{attribute addProperty BoxType "EL2258-0000-0016"}
{attribute addProperty Id "MTO_Inputs_ChannelAT %I*ARRAY[0..7] OF MTO_Inputs_Channel_5AD475AF8721090MTO_Outputs_10x_ChannelAT %Q*ARRAY[0..7] OF MTO_Outputs_10x_Channel_4C67AB5F45845730WcStateAT %I*WcState_F855686C1620InfoDataAT %I*InfoData_0BDED7BF144180"}
{attribute addProperty CRC "3021902586"}
{attribute addProperty SizeInBites "5616"}
{attribute addProperty SizeInBytes "702"}
TYPE EL2258_9EFD418A :
STRUCT
	{attribute addProperty Name "MTO_Inputs_Channel"}
	MTO_Inputs_Channel : ARRAY[0..7] OF MTO_Inputs_Channel_5AD475AF;
	{attribute addProperty Name "MTO_Outputs_10x_Channel"}
	MTO_Outputs_10x_Channel : ARRAY[0..7] OF MTO_Outputs_10x_Channel_4C67AB5F;
	{attribute addProperty Name "WcState"}
	WcState : WcState_F855686C;
	{attribute addProperty Name "InfoData"}
	InfoData : InfoData_0BDED7BF;
END_STRUCT
END_TYPE

(* stored: Version 1.2.0.0, ProductVersion 3.1.4024.9
   DUT EL2258_9EFD418A: Id {49d70f5d-97dc-48b7-b338-2fde3e451101} *)
